FUNCTION Convert_BOOL_TO_USINT : BOOL
VAR_INPUT
	in : BOOL;
	out : REFERENCE TO USINT;
END_VAR

out := BOOL_TO_USINT(in);
Convert_BOOL_TO_USINT := TRUE;

END_FUNCTION

(* stored: Version 1.1.0.1, ProductVersion 3.1.4024.12
   POU Convert_BOOL_TO_USINT: Id {cb4c7d0f-9f6e-4a21-80b1-2a7a48b4b5a2}, SpecialFunc None *)
